INTERFACE I_LinkDestination

PROPERTY PUBLIC Connected : BOOL
GET
END_GET
END_PROPERTY

PROPERTY PUBLIC Data : I_Datatype
GET
END_GET
END_PROPERTY

METHOD PUBLIC Disconnect
END_METHOD

PROPERTY PUBLIC Name : T_MAXSTRING
GET
END_GET
END_PROPERTY

METHOD PUBLIC TryConnectTo : BOOL
VAR_INPUT
	Source : I_LinkSource;
END_VAR
END_METHOD

END_INTERFACE

(* stored: Version 1.1.0.1, ProductVersion 3.1.4024.13
   Itf I_LinkDestination: Id {47d6d751-c45c-0a11-25d5-a90b9e650bea}
   Property Connected: Id {274512c4-02cb-0fc3-2098-48b07c51d71a}
   Get Get: Id {a8a90f64-4723-03d5-17bf-5c3881807787}
   Property Data: Id {bb92110f-6a47-01db-360f-a5e3eb7309d8}
   Get Get: Id {fa5eed5a-6233-0e38-35c5-aed04667af8f}
   Method Disconnect: Id {2f84ecf4-40b9-05e0-3fef-85bc181022be}
   Property Name: Id {3bfb0383-db68-023e-2e6e-e41c5a765cd0}
   Get Get: Id {9e3db619-f544-07bd-1879-79e5d12728e1}
   Method TryConnectTo: Id {9c3c5c90-8dba-0e4f-3c00-1348fe633275} *)
